// TIA Portal V18 export
// export: Created 2026-06-22T12:39:26.0576196Z, ExportSetting WithDefaults, DisplayName Totally Integrated Automation Portal, DisplayVersion V18, DisplayName TIA Portal Openness, DisplayVersion V18, DisplayName TIA Portal Version Control Interface, DisplayVersion V18, DisplayName STEP 7 Professional, DisplayVersion V18, DisplayName STEP 7 Safety, DisplayVersion V18, DisplayName WinCC Professional, DisplayVersion V18
TagTable "Default tag table"
  Logged_In : Int  (1 s)
  HMI_SP_PLC2_Nhiet_Do_Bon4 : Real  (PLC tag HMI_SP_PLC2_Nhiet_Do_Bon4, HMI_Connection_1, 1 s)
  HMI_SP_PLC2_Nuoc_Bon3 : Real  (PLC tag HMI_SP_PLC2_Nuoc_Bon3, HMI_Connection_1, 1 s)
